// SIMATIC S7-200 SMART project (STEP 7-Micro/WIN SMART), CPU ST40

ORGANIZATION_BLOCK MAIN:OB1
TITLE=程序注释
BEGIN
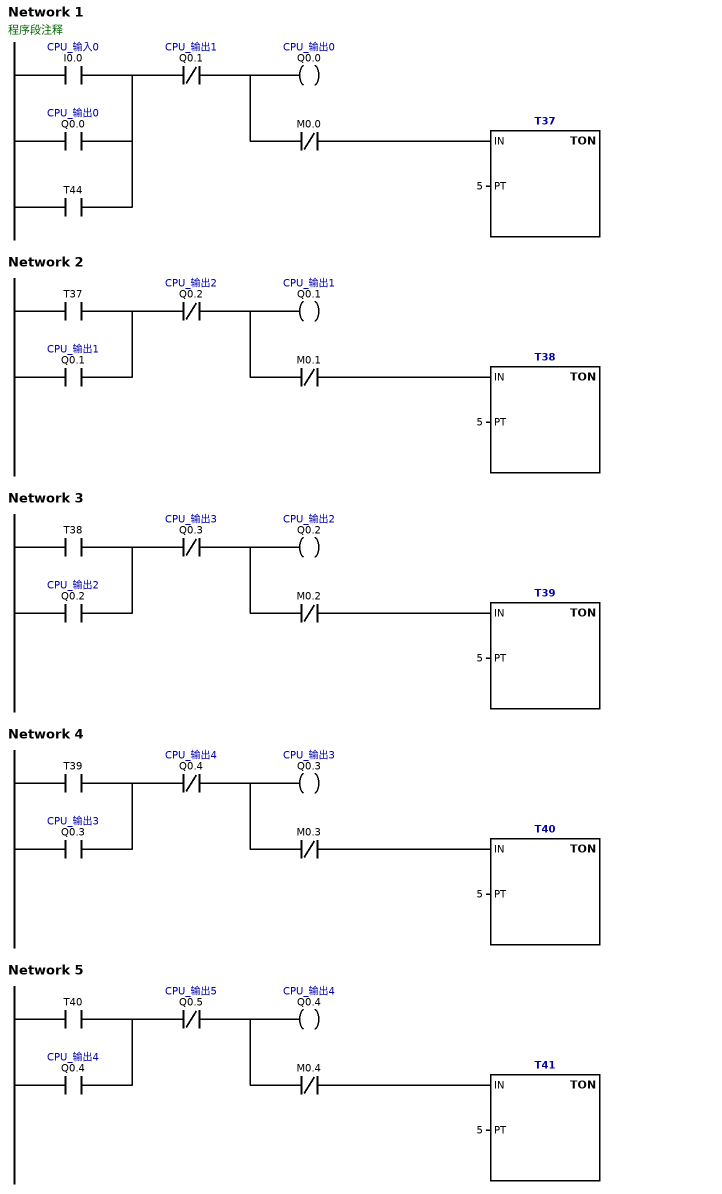
Network 1
// 程序段注释
LD     CPU_输入0:I0.0
O      CPU_输出0:Q0.0
O      T44
AN     CPU_输出1:Q0.1
=      CPU_输出0:Q0.0
AN     M0.0
TON    T37, 5
Network 2
LD     T37
O      CPU_输出1:Q0.1
AN     CPU_输出2:Q0.2
=      CPU_输出1:Q0.1
AN     M0.1
TON    T38, 5
Network 3
LD     T38
O      CPU_输出2:Q0.2
AN     CPU_输出3:Q0.3
=      CPU_输出2:Q0.2
AN     M0.2
TON    T39, 5
Network 4
LD     T39
O      CPU_输出3:Q0.3
AN     CPU_输出4:Q0.4
=      CPU_输出3:Q0.3
AN     M0.3
TON    T40, 5
Network 5
LD     T40
O      CPU_输出4:Q0.4
AN     CPU_输出5:Q0.5
=      CPU_输出4:Q0.4
AN     M0.4
TON    T41, 5
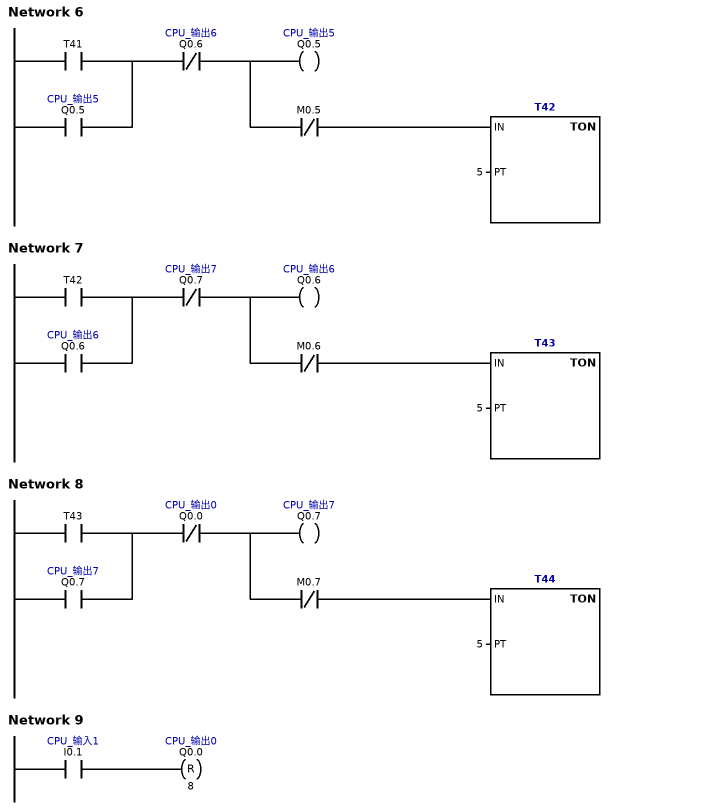
Network 6
LD     T41
O      CPU_输出5:Q0.5
AN     CPU_输出6:Q0.6
=      CPU_输出5:Q0.5
AN     M0.5
TON    T42, 5
Network 7
LD     T42
O      CPU_输出6:Q0.6
AN     CPU_输出7:Q0.7
=      CPU_输出6:Q0.6
AN     M0.6
TON    T43, 5
Network 8
LD     T43
O      CPU_输出7:Q0.7
AN     CPU_输出0:Q0.0
=      CPU_输出7:Q0.7
AN     M0.7
TON    T44, 5
Network 9
LD     CPU_输入1:I0.1
R      CPU_输出0:Q0.0, 8
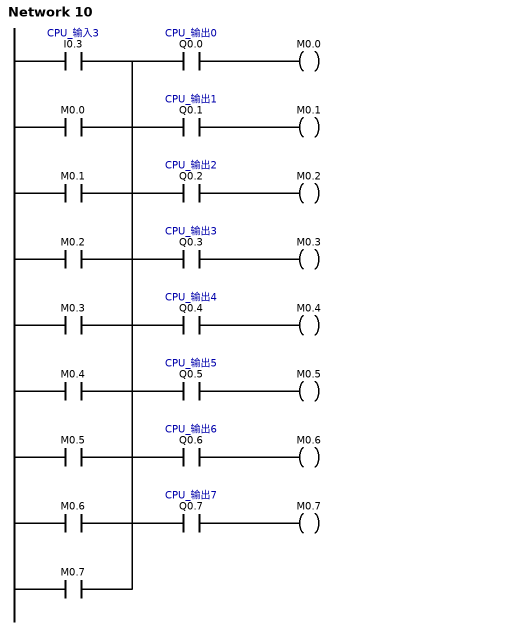
Network 10
LD     CPU_输入3:I0.3
O      M0.0
O      M0.1
O      M0.2
O      M0.3
O      M0.4
O      M0.5
O      M0.6
O      M0.7
LPS
A      CPU_输出0:Q0.0
=      M0.0
LRD
A      CPU_输出1:Q0.1
=      M0.1
LRD
A      CPU_输出2:Q0.2
=      M0.2
LRD
A      CPU_输出3:Q0.3
=      M0.3
LRD
A      CPU_输出4:Q0.4
=      M0.4
LRD
A      CPU_输出5:Q0.5
=      M0.5
LRD
A      CPU_输出6:Q0.6
=      M0.6
LPP
A      CPU_输出7:Q0.7
=      M0.7
END_ORGANIZATION_BLOCK
